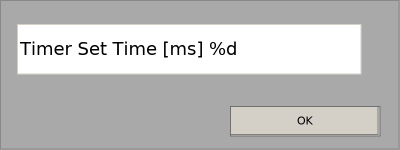
VISUALIZATION DialogTimer_ValveClose  // 400x150
    Button (230,106 150x30), "OK"
        OnMouseClick: CloseDialog Dialog=DialogTimer_ValveClose, Result=OK, NumpadKeypadSet=True
    Textfield (17,24 344x50), "Timer Set Time [ms] %d", text variable: PersistentStruct.TimerPressUp
        OnMouseClick: write the text variable via Edit
END_VISUALIZATION

(* stored: Version 1.1.0.1, ProductVersion 3.1.4024.3
   Visu DialogTimer_ValveClose: Id {3ca96a82-6667-4ee9-b8e8-a44f924f2ae1} *)
